(* IEC 61131-3 sources: sphere-usecases/sector-energy/olmsted-hydro/implementations/openplc/st/legacy, 2 files *)

(* ---- ps_hydro_controller.st ---- *)
(*
 * SPHERE Power Systems - Generic Hydro Station Controller
 * IEC 61131-3 Structured Text for OpenPLC
 *
 * Control state machine for hydro power generation:
 *   IDLE -> STARTUP -> RUNNING -> SHUTDOWN -> IDLE
 *                  \-> TRIPPED (on any trip) -> IDLE (after reset)
 *
 * This program runs on the CONTROLLER PLC and implements:
 *   - State machine for unit operation
 *   - Permissive checks for startup
 *   - Power tracking via gate modulation (P-control)
 *   - Trip detection and response
 *   - Mismatch alarm generation
 *
 * Inputs (from HMI):
 *   - Start, Stop, Reset commands (%IX0.0-0.2)
 *   - Mode Auto, Run Enable (%IX0.3-0.4)
 *
 * Inputs (from Simulator via bridge):
 *   - Gate position, sensors (%IW70-77)
 *   - Breaker/Spill status (%IX2.0-2.1)
 *
 * Outputs (to Simulator via bridge):
 *   - Gate command (%QW100)
 *   - Breaker/Spill commands (%QX5.0-5.1)
 *
 * Outputs (to HMI):
 *   - State indicators (%QX7.0-7.5)
 *   - Trip indicators (%QX8.0-8.3)
 *   - Alarm indicators (%QX9.0-9.2)
 *)

(* ═══════════════════════════════════════════════════════════════════════════
   GLOBAL VARIABLES - I/O MAPPING
   ═══════════════════════════════════════════════════════════════════════════ *)
VAR_GLOBAL
    (* HMI Inputs *)
    in_Start_Cmd AT %IX0.0 : BOOL;      (* Start pushbutton *)
    in_Stop_Cmd AT %IX0.1 : BOOL;       (* Stop pushbutton *)
    in_Reset_Cmd AT %IX0.2 : BOOL;      (* Trip reset pushbutton *)
    in_Mode_Auto AT %IX0.3 : BOOL;      (* Auto mode enable *)
    in_Run_Enable AT %IX0.4 : BOOL;     (* Run permissive *)

    (* Power setpoint - could come from HMI or external *)
    in_Power_Setpoint AT %IW60 : INT;   (* 0-1000 = 0-100 MW *)

    (* Process Inputs from Simulator (via bridge) *)
    in_Gate_Pos AT %IW70 : INT;         (* Gate position 0-1000 = 0-100% *)
    in_Res_Level AT %IW71 : INT;        (* Reservoir level 0-3000 = 0-30.00 m *)
    in_Head AT %IW72 : INT;             (* Head 0-1500 = 0-150.0 m *)
    in_Flow AT %IW73 : INT;             (* Flow 0-1500 = 0-150.0 m3/s *)
    in_Pressure AT %IW74 : INT;         (* Pressure kPa *)
    in_Speed_Pct AT %IW75 : INT;        (* Speed 0-1500 = 0-150.0% *)
    in_Freq_Hz AT %IW76 : INT;          (* Frequency 5500-6500 = 55-65 Hz *)
    in_Power_MW AT %IW77 : INT;         (* Power 0-1000 = 0-100 MW *)

    in_Breaker_Sts AT %IX2.0 : BOOL;    (* Breaker closed status *)
    in_Spill_Sts AT %IX2.1 : BOOL;      (* Spillway open status *)

    (* Actuator Outputs to Simulator (via bridge) *)
    out_Gate_Cmd AT %QW100 : INT;       (* Gate command 0-1000 = 0-100% *)
    out_Power_Setpoint AT %QW101 : INT; (* Power setpoint passthrough *)
    out_Breaker_Cmd AT %QX5.0 : BOOL;   (* Breaker close command *)
    out_Spill_Cmd AT %QX5.1 : BOOL;     (* Spillway open command *)

    (* State Outputs to HMI *)
    out_State_Idle AT %QX7.0 : BOOL;
    out_State_Startup AT %QX7.1 : BOOL;
    out_State_Running AT %QX7.2 : BOOL;
    out_State_Shutdown AT %QX7.3 : BOOL;
    out_State_Tripped AT %QX7.4 : BOOL;
    out_Permissives_Ready AT %QX7.5 : BOOL;

    (* Trip Outputs *)
    out_Trip_Overspeed AT %QX8.0 : BOOL;
    out_Trip_Overpressure AT %QX8.1 : BOOL;
    out_Trip_LowHead AT %QX8.2 : BOOL;
    out_Trip_Manual AT %QX8.3 : BOOL;

    (* Alarm Outputs *)
    out_Alarm_GateMismatch AT %QX9.0 : BOOL;
    out_Alarm_BreakerMismatch AT %QX9.1 : BOOL;
    out_Alarm_LowLevel AT %QX9.2 : BOOL;
END_VAR

(* ═══════════════════════════════════════════════════════════════════════════
   MAIN PROGRAM
   ═══════════════════════════════════════════════════════════════════════════ *)
PROGRAM HydroController
VAR
    (* ─── State Machine ──────────────────────────────────────────────────── *)
    State : INT := 0;                   (* 0=IDLE, 1=STARTUP, 2=RUNNING, 3=SHUTDOWN, 4=TRIPPED *)
    STATE_IDLE : INT := 0;
    STATE_STARTUP : INT := 1;
    STATE_RUNNING : INT := 2;
    STATE_SHUTDOWN : INT := 3;
    STATE_TRIPPED : INT := 4;

    (* ─── Permissives ────────────────────────────────────────────────────── *)
    Perm_Level_OK : BOOL := FALSE;      (* Reservoir level adequate *)
    Perm_Head_OK : BOOL := FALSE;       (* Head above minimum *)
    Perm_No_Trips : BOOL := FALSE;      (* No active trips *)
    Perm_Run_Enable : BOOL := FALSE;    (* Operator run enable *)
    All_Permissives : BOOL := FALSE;    (* Combined permissive *)

    (* ─── Trip Latches ───────────────────────────────────────────────────── *)
    Trip_Overspeed_Latch : BOOL := FALSE;
    Trip_Overpressure_Latch : BOOL := FALSE;
    Trip_LowHead_Latch : BOOL := FALSE;
    Trip_Manual_Latch : BOOL := FALSE;
    Any_Trip : BOOL := FALSE;

    (* ─── Control Parameters ─────────────────────────────────────────────── *)
    No_Load_Gate_Pct : REAL := 5.0;     (* Gate position for no-load sync *)
    Sync_Speed_Low : REAL := 99.0;      (* Min speed for sync % *)
    Sync_Speed_High : REAL := 101.0;    (* Max speed for sync % *)
    Min_Power_MW : REAL := 1.0;         (* Min power before breaker open *)
    Kp_Gate : REAL := 2.0;              (* Power control gain *)
    Gate_Shutdown_Rate : REAL := 5.0;   (* %/sample during shutdown *)
    Gate_Emerg_Rate : REAL := 20.0;     (* %/sample during trip *)

    (* ─── Trip Thresholds ────────────────────────────────────────────────── *)
    Overspeed_Trip_Pct : REAL := 110.0;
    Overpressure_Trip_kPa : REAL := 1500.0;
    Min_Head_m : REAL := 10.0;
    Low_Level_m : REAL := 8.0;          (* Alarm threshold *)

    (* ─── Mismatch Alarm Parameters ──────────────────────────────────────── *)
    Gate_Mismatch_Pct : REAL := 5.0;    (* Alarm if error > 5% *)
    Gate_Mismatch_Delay : INT := 50;    (* 5 sec at 100ms cycle *)
    Breaker_Mismatch_Delay : INT := 5;  (* 0.5 sec *)
    Gate_Mismatch_Timer : INT := 0;
    Breaker_Mismatch_Timer : INT := 0;

    (* ─── Process Values (scaled) ────────────────────────────────────────── *)
    Gate_Pos_Pct : REAL;
    Gate_Cmd_Pct : REAL := 0.0;
    Res_Level_m : REAL;
    Head_m : REAL;
    Flow_m3s : REAL;
    Pressure_kPa : REAL;
    Speed_Pct : REAL;
    Freq_Hz : REAL;
    Power_MW : REAL;
    Power_Setpoint_MW : REAL;

    (* ─── Control Calculations ───────────────────────────────────────────── *)
    Power_Error : REAL;
    Gate_Adjustment : REAL;

    (* ─── Edge Detection ─────────────────────────────────────────────────── *)
    Start_Cmd_Prev : BOOL := FALSE;
    Stop_Cmd_Prev : BOOL := FALSE;
    Reset_Cmd_Prev : BOOL := FALSE;
    Start_Rising : BOOL := FALSE;
    Stop_Rising : BOOL := FALSE;
    Reset_Rising : BOOL := FALSE;
END_VAR

(* ═══════════════════════════════════════════════════════════════════════════
   CONTROL LOGIC
   ═══════════════════════════════════════════════════════════════════════════ *)

(* ─── 1. SCALE INPUTS ─────────────────────────────────────────────────────── *)
Gate_Pos_Pct := INT_TO_REAL(in_Gate_Pos) / 10.0;
Res_Level_m := INT_TO_REAL(in_Res_Level) / 100.0;
Head_m := INT_TO_REAL(in_Head) / 10.0;
Flow_m3s := INT_TO_REAL(in_Flow) / 10.0;
Pressure_kPa := INT_TO_REAL(in_Pressure);
Speed_Pct := INT_TO_REAL(in_Speed_Pct) / 10.0;
Freq_Hz := INT_TO_REAL(in_Freq_Hz) / 100.0;
Power_MW := INT_TO_REAL(in_Power_MW) / 10.0;
Power_Setpoint_MW := INT_TO_REAL(in_Power_Setpoint) / 10.0;

(* ─── 2. EDGE DETECTION FOR COMMANDS ──────────────────────────────────────── *)
Start_Rising := in_Start_Cmd AND NOT Start_Cmd_Prev;
Stop_Rising := in_Stop_Cmd AND NOT Stop_Cmd_Prev;
Reset_Rising := in_Reset_Cmd AND NOT Reset_Cmd_Prev;
Start_Cmd_Prev := in_Start_Cmd;
Stop_Cmd_Prev := in_Stop_Cmd;
Reset_Cmd_Prev := in_Reset_Cmd;

(* ─── 3. TRIP DETECTION ───────────────────────────────────────────────────── *)
(* Check trip conditions and latch *)
IF Speed_Pct > Overspeed_Trip_Pct THEN
    Trip_Overspeed_Latch := TRUE;
END_IF;

IF Pressure_kPa > Overpressure_Trip_kPa THEN
    Trip_Overpressure_Latch := TRUE;
END_IF;

IF Head_m < Min_Head_m AND State = STATE_RUNNING THEN
    Trip_LowHead_Latch := TRUE;
END_IF;

(* Manual trip via Stop during running with specific pattern *)
(* For now, no separate manual trip - Stop just initiates shutdown *)

(* Combined trip check *)
Any_Trip := Trip_Overspeed_Latch OR Trip_Overpressure_Latch OR
            Trip_LowHead_Latch OR Trip_Manual_Latch;

(* ─── 4. PERMISSIVE CHECKS ────────────────────────────────────────────────── *)
Perm_Level_OK := Res_Level_m > Low_Level_m;
Perm_Head_OK := Head_m >= Min_Head_m;
Perm_No_Trips := NOT Any_Trip;
Perm_Run_Enable := in_Run_Enable;

All_Permissives := Perm_Level_OK AND Perm_Head_OK AND
                   Perm_No_Trips AND Perm_Run_Enable;

(* ─── 5. STATE MACHINE ────────────────────────────────────────────────────── *)
CASE State OF
    (* ═══ IDLE STATE ═══ *)
    0: (* STATE_IDLE *)
        (* Outputs: gate closed, breaker open *)
        Gate_Cmd_Pct := 0.0;
        out_Breaker_Cmd := FALSE;
        out_Spill_Cmd := FALSE;

        (* Transitions *)
        IF Start_Rising AND All_Permissives THEN
            State := STATE_STARTUP;
        END_IF;

    (* ═══ STARTUP STATE ═══ *)
    1: (* STATE_STARTUP *)
        (* Ramp gate to no-load position *)
        IF Gate_Cmd_Pct < No_Load_Gate_Pct THEN
            Gate_Cmd_Pct := Gate_Cmd_Pct + 1.0;  (* Ramp up 1%/cycle *)
        ELSE
            Gate_Cmd_Pct := No_Load_Gate_Pct;
        END_IF;

        (* Check for sync conditions *)
        IF Speed_Pct >= Sync_Speed_Low AND Speed_Pct <= Sync_Speed_High THEN
            (* Close breaker when speed is in sync range *)
            out_Breaker_Cmd := TRUE;

            (* Transition to running when breaker closes *)
            IF in_Breaker_Sts THEN
                State := STATE_RUNNING;
            END_IF;
        END_IF;

        (* Trip handling *)
        IF Any_Trip THEN
            State := STATE_TRIPPED;
        END_IF;

        (* Stop command *)
        IF Stop_Rising THEN
            State := STATE_SHUTDOWN;
        END_IF;

    (* ═══ RUNNING STATE ═══ *)
    2: (* STATE_RUNNING *)
        (* Power tracking via P-control *)
        Power_Error := Power_Setpoint_MW - Power_MW;
        Gate_Adjustment := Kp_Gate * Power_Error;

        (* Apply adjustment with limits *)
        Gate_Cmd_Pct := Gate_Cmd_Pct + Gate_Adjustment;

        (* Clamp gate command *)
        IF Gate_Cmd_Pct < 0.0 THEN Gate_Cmd_Pct := 0.0; END_IF;
        IF Gate_Cmd_Pct > 100.0 THEN Gate_Cmd_Pct := 100.0; END_IF;

        (* Breaker stays closed *)
        out_Breaker_Cmd := TRUE;

        (* Trip handling - immediate transition *)
        IF Any_Trip THEN
            State := STATE_TRIPPED;
        END_IF;

        (* Stop command - normal shutdown *)
        IF Stop_Rising THEN
            State := STATE_SHUTDOWN;
        END_IF;

    (* ═══ SHUTDOWN STATE ═══ *)
    3: (* STATE_SHUTDOWN *)
        (* Ramp gate down *)
        Gate_Cmd_Pct := Gate_Cmd_Pct - Gate_Shutdown_Rate;
        IF Gate_Cmd_Pct < 0.0 THEN
            Gate_Cmd_Pct := 0.0;
        END_IF;

        (* Open breaker when power is low enough *)
        IF Power_MW < Min_Power_MW THEN
            out_Breaker_Cmd := FALSE;
        END_IF;

        (* Transition to idle when gate closed and breaker open *)
        IF Gate_Cmd_Pct <= 0.0 AND NOT in_Breaker_Sts THEN
            State := STATE_IDLE;
        END_IF;

        (* Trip can still occur during shutdown *)
        IF Any_Trip THEN
            State := STATE_TRIPPED;
        END_IF;

    (* ═══ TRIPPED STATE ═══ *)
    4: (* STATE_TRIPPED *)
        (* Emergency actions *)
        out_Breaker_Cmd := FALSE;           (* Open breaker immediately *)

        (* Fast gate close *)
        Gate_Cmd_Pct := Gate_Cmd_Pct - Gate_Emerg_Rate;
        IF Gate_Cmd_Pct < 0.0 THEN
            Gate_Cmd_Pct := 0.0;
        END_IF;

        (* Open spillway on overspeed to dump water *)
        IF Trip_Overspeed_Latch THEN
            out_Spill_Cmd := TRUE;
        END_IF;

        (* Reset handling - only when gate closed and breaker open *)
        IF Reset_Rising AND Gate_Cmd_Pct <= 0.0 AND NOT in_Breaker_Sts THEN
            (* Clear all trip latches *)
            Trip_Overspeed_Latch := FALSE;
            Trip_Overpressure_Latch := FALSE;
            Trip_LowHead_Latch := FALSE;
            Trip_Manual_Latch := FALSE;

            (* Close spillway *)
            out_Spill_Cmd := FALSE;

            (* Return to idle *)
            State := STATE_IDLE;
        END_IF;

END_CASE;

(* ─── 6. MISMATCH ALARM LOGIC ─────────────────────────────────────────────── *)
(* Gate mismatch alarm *)
IF ABS(Gate_Cmd_Pct - Gate_Pos_Pct) > Gate_Mismatch_Pct THEN
    Gate_Mismatch_Timer := Gate_Mismatch_Timer + 1;
    IF Gate_Mismatch_Timer >= Gate_Mismatch_Delay THEN
        out_Alarm_GateMismatch := TRUE;
    END_IF;
ELSE
    Gate_Mismatch_Timer := 0;
    out_Alarm_GateMismatch := FALSE;
END_IF;

(* Breaker mismatch alarm *)
IF out_Breaker_Cmd <> in_Breaker_Sts THEN
    Breaker_Mismatch_Timer := Breaker_Mismatch_Timer + 1;
    IF Breaker_Mismatch_Timer >= Breaker_Mismatch_Delay THEN
        out_Alarm_BreakerMismatch := TRUE;
    END_IF;
ELSE
    Breaker_Mismatch_Timer := 0;
    out_Alarm_BreakerMismatch := FALSE;
END_IF;

(* Low level alarm *)
out_Alarm_LowLevel := Res_Level_m < Low_Level_m;

(* ─── 7. WRITE OUTPUTS ────────────────────────────────────────────────────── *)
(* Scale and write gate command *)
out_Gate_Cmd := REAL_TO_INT(Gate_Cmd_Pct * 10.0);

(* Pass through power setpoint *)
out_Power_Setpoint := in_Power_Setpoint;

(* State indicators *)
out_State_Idle := (State = STATE_IDLE);
out_State_Startup := (State = STATE_STARTUP);
out_State_Running := (State = STATE_RUNNING);
out_State_Shutdown := (State = STATE_SHUTDOWN);
out_State_Tripped := (State = STATE_TRIPPED);
out_Permissives_Ready := All_Permissives;

(* Trip indicators *)
out_Trip_Overspeed := Trip_Overspeed_Latch;
out_Trip_Overpressure := Trip_Overpressure_Latch;
out_Trip_LowHead := Trip_LowHead_Latch;
out_Trip_Manual := Trip_Manual_Latch;

END_PROGRAM

(* ---- ps_hydro_simulator.st ---- *)
(*
 * SPHERE Power Systems - Generic Hydro Station Simulator
 * IEC 61131-3 Structured Text for OpenPLC
 *
 * Physics model for hydro power generation:
 *   Reservoir -> Penstock -> Wicket Gate -> Turbine -> Generator -> Breaker -> Grid
 *
 * This program runs on the SIMULATOR PLC and models:
 *   - Reservoir mass balance with head calculation
 *   - Penstock flow dynamics (1st-order lag)
 *   - Wicket gate actuator with slew limits
 *   - Turbine/generator power conversion
 *   - Breaker dynamics
 *   - Trip condition detection
 *
 * Inputs (from Controller via bridge):
 *   - Gate command (%IW200)
 *   - Breaker command (%IX3.0)
 *   - Spill command (%IX3.1)
 *
 * Outputs (to Controller via bridge):
 *   - Gate position (%QW300)
 *   - Reservoir level, head, flow, pressure, speed, freq, power (%QW301-307)
 *   - Breaker status, spill status (%QX40.0-40.1)
 *)

(* ═══════════════════════════════════════════════════════════════════════════
   GLOBAL VARIABLES - I/O MAPPING
   ═══════════════════════════════════════════════════════════════════════════ *)
VAR_GLOBAL
    (* Inputs from Controller (via bridge) *)
    in_Gate_Cmd AT %IW200 : INT;        (* Gate command 0-1000 = 0-100% *)
    in_Breaker_Cmd AT %IX3.0 : BOOL;    (* Breaker close command *)
    in_Spill_Cmd AT %IX3.1 : BOOL;      (* Spillway open command *)

    (* Outputs to Controller (via bridge) *)
    out_Gate_Pos AT %QW300 : INT;       (* Gate position 0-1000 = 0-100% *)
    out_Res_Level AT %QW301 : INT;      (* Reservoir level 0-3000 = 0-30.00 m *)
    out_Head AT %QW302 : INT;           (* Head 0-1500 = 0-150.0 m *)
    out_Flow AT %QW303 : INT;           (* Flow 0-1500 = 0-150.0 m3/s *)
    out_Pressure AT %QW304 : INT;       (* Pressure 0-2000 kPa *)
    out_Speed_Pct AT %QW305 : INT;      (* Speed 0-1500 = 0-150.0% *)
    out_Freq_Hz AT %QW306 : INT;        (* Frequency 5500-6500 = 55.00-65.00 Hz *)
    out_Power_MW AT %QW307 : INT;       (* Power 0-1000 = 0-100.0 MW *)

    out_Breaker_Sts AT %QX40.0 : BOOL;  (* Breaker closed status *)
    out_Spill_Sts AT %QX40.1 : BOOL;    (* Spillway open status *)
END_VAR

(* ═══════════════════════════════════════════════════════════════════════════
   MAIN PROGRAM
   ═══════════════════════════════════════════════════════════════════════════ *)
PROGRAM HydroSimulator
VAR
    (* ─── Physical Parameters (from profile) ─────────────────────────────── *)
    (* Reservoir *)
    Res_Area_m2 : REAL := 10000.0;      (* Reservoir surface area *)
    Res_Level_m : REAL := 20.0;         (* Current reservoir level *)
    Res_Inflow_m3s : REAL := 50.0;      (* Natural inflow *)
    Res_Min_m : REAL := 5.0;            (* Minimum operating level *)
    Res_Max_m : REAL := 25.0;           (* Maximum level *)
    Tailwater_m : REAL := 0.0;          (* Tailwater elevation *)

    (* Penstock *)
    Penstock_Tau_sec : REAL := 5.0;     (* Flow inertia time constant *)
    Static_Head_m : REAL := 100.0;      (* Reference static head *)

    (* Turbine *)
    Q_Max_m3s : REAL := 100.0;          (* Maximum flow capacity *)
    Eta_Turbine : REAL := 0.90;         (* Turbine efficiency *)
    K_Q : REAL := 10.0;                 (* Flow coefficient *)

    (* Generator *)
    Eta_Gen : REAL := 0.97;             (* Generator efficiency *)
    P_Rated_MW : REAL := 80.0;          (* Rated power *)
    Inertia_H : REAL := 4.0;            (* Inertia constant (seconds) *)
    Sync_Speed_Pct : REAL := 100.0;     (* Synchronous speed reference *)

    (* Gate actuator *)
    Gate_Travel_sec : REAL := 10.0;     (* Full stroke time *)
    Gate_Slew_Max : REAL := 10.0;       (* Max slew rate %/s *)
    Gate_Tau_sec : REAL := 1.0;         (* Servo time constant *)
    Gate_Emerg_sec : REAL := 3.0;       (* Emergency close time *)

    (* Breaker *)
    Breaker_Open_sec : REAL := 0.06;    (* Open time *)
    Breaker_Close_sec : REAL := 0.05;   (* Close time *)

    (* Spillway *)
    Spill_Open_sec : REAL := 5.0;       (* Spillway open time *)

    (* Physical constants *)
    RHO : REAL := 1000.0;               (* Water density kg/m3 *)
    G : REAL := 9.81;                   (* Gravity m/s2 *)

    (* ─── State Variables ────────────────────────────────────────────────── *)
    Gate_Pos_Pct : REAL := 0.0;         (* Actual gate position % *)
    Gate_Vel : REAL := 0.0;             (* Gate velocity %/s *)
    Flow_m3s : REAL := 0.0;             (* Actual flow rate *)
    Flow_Target_m3s : REAL := 0.0;      (* Target flow (gate opening) *)
    Head_m : REAL := 100.0;             (* Net hydraulic head *)
    Pressure_kPa : REAL := 981.0;       (* Penstock pressure *)
    Speed_Pct : REAL := 0.0;            (* Turbine speed % of sync *)
    Freq_Hz : REAL := 0.0;              (* Electrical frequency *)
    P_Mech_MW : REAL := 0.0;            (* Mechanical power *)
    P_Elec_MW : REAL := 0.0;            (* Electrical power *)

    Breaker_Closed : BOOL := FALSE;     (* Breaker state *)
    Breaker_Timer : REAL := 0.0;        (* Breaker transition timer *)
    Spill_Open : BOOL := FALSE;         (* Spillway state *)
    Spill_Timer : REAL := 0.0;          (* Spillway transition timer *)

    (* ─── Intermediate Calculations ──────────────────────────────────────── *)
    Gate_Cmd_Pct : REAL;                (* Commanded gate position % *)
    Gate_Error : REAL;                  (* Gate position error *)
    dQ_dt : REAL;                       (* Flow rate of change *)
    dLevel_dt : REAL;                   (* Level rate of change *)
    dSpeed_dt : REAL;                   (* Speed rate of change *)
    P_Load_MW : REAL;                   (* Grid load (when connected) *)
    Spill_Flow_m3s : REAL;              (* Spillway discharge *)

    (* ─── Timing ─────────────────────────────────────────────────────────── *)
    DT : REAL := 0.1;                   (* Simulation timestep (100ms) *)

    (* ─── Trip Detection ─────────────────────────────────────────────────── *)
    Overspeed : BOOL := FALSE;
    Overpressure : BOOL := FALSE;
    LowHead : BOOL := FALSE;
END_VAR

(* ═══════════════════════════════════════════════════════════════════════════
   SIMULATION LOGIC
   ═══════════════════════════════════════════════════════════════════════════ *)

(* ─── 1. PROCESS INPUTS ───────────────────────────────────────────────────── *)
(* Convert scaled integer inputs to engineering units *)
Gate_Cmd_Pct := INT_TO_REAL(in_Gate_Cmd) / 10.0;  (* 0-1000 -> 0-100% *)

(* Clamp command to valid range *)
IF Gate_Cmd_Pct < 0.0 THEN Gate_Cmd_Pct := 0.0; END_IF;
IF Gate_Cmd_Pct > 100.0 THEN Gate_Cmd_Pct := 100.0; END_IF;

(* ─── 2. GATE ACTUATOR DYNAMICS ───────────────────────────────────────────── *)
(* First-order servo response with slew limiting *)
Gate_Error := Gate_Cmd_Pct - Gate_Pos_Pct;
Gate_Vel := Gate_Error / Gate_Tau_sec;

(* Apply slew rate limits *)
IF Gate_Vel > Gate_Slew_Max THEN
    Gate_Vel := Gate_Slew_Max;
ELSIF Gate_Vel < -Gate_Slew_Max THEN
    Gate_Vel := -Gate_Slew_Max;
END_IF;

(* Integrate gate position *)
Gate_Pos_Pct := Gate_Pos_Pct + Gate_Vel * DT;

(* Clamp to physical limits *)
IF Gate_Pos_Pct < 0.0 THEN Gate_Pos_Pct := 0.0; END_IF;
IF Gate_Pos_Pct > 100.0 THEN Gate_Pos_Pct := 100.0; END_IF;

(* ─── 3. RESERVOIR MASS BALANCE ───────────────────────────────────────────── *)
(* Calculate spillway flow if open *)
IF Spill_Open THEN
    (* Simple spillway model: proportional to level above threshold *)
    IF Res_Level_m > 22.0 THEN
        Spill_Flow_m3s := 20.0 * (Res_Level_m - 22.0);
    ELSE
        Spill_Flow_m3s := 0.0;
    END_IF;
ELSE
    Spill_Flow_m3s := 0.0;
END_IF;

(* Mass balance: dV/dt = Q_in - Q_turbine - Q_spill *)
dLevel_dt := (Res_Inflow_m3s - Flow_m3s - Spill_Flow_m3s) / Res_Area_m2;
Res_Level_m := Res_Level_m + dLevel_dt * DT;

(* Clamp reservoir level *)
IF Res_Level_m < 0.0 THEN Res_Level_m := 0.0; END_IF;
IF Res_Level_m > Res_Max_m THEN Res_Level_m := Res_Max_m; END_IF;

(* Calculate net head: H = reservoir_level - tailwater *)
Head_m := Res_Level_m + Static_Head_m - Tailwater_m;
IF Head_m < 0.0 THEN Head_m := 0.0; END_IF;

(* ─── 4. PENSTOCK FLOW DYNAMICS ───────────────────────────────────────────── *)
(* Target flow based on gate opening and head *)
(* Q = k_q * (gate_pos/100) * sqrt(H) *)
IF Head_m > 0.0 THEN
    Flow_Target_m3s := K_Q * (Gate_Pos_Pct / 100.0) * SQRT(Head_m);
ELSE
    Flow_Target_m3s := 0.0;
END_IF;

(* Limit to maximum flow *)
IF Flow_Target_m3s > Q_Max_m3s THEN
    Flow_Target_m3s := Q_Max_m3s;
END_IF;

(* First-order lag for flow inertia: dQ/dt = (Q_target - Q) / tau *)
dQ_dt := (Flow_Target_m3s - Flow_m3s) / Penstock_Tau_sec;
Flow_m3s := Flow_m3s + dQ_dt * DT;

(* Clamp flow *)
IF Flow_m3s < 0.0 THEN Flow_m3s := 0.0; END_IF;

(* Calculate penstock pressure: P = rho * g * H *)
Pressure_kPa := RHO * G * Head_m / 1000.0;

(* Check for water hammer (rapid flow change) *)
IF ABS(dQ_dt) > 20.0 THEN
    (* Approximate pressure surge *)
    Pressure_kPa := Pressure_kPa * 1.5;
END_IF;

(* ─── 5. TURBINE/GENERATOR DYNAMICS ───────────────────────────────────────── *)
(* Mechanical power: P_mech = rho * g * Q * H * eta_t *)
P_Mech_MW := RHO * G * Flow_m3s * Head_m * Eta_Turbine / 1000000.0;

(* Speed dynamics depend on breaker state *)
IF Breaker_Closed THEN
    (* Connected to grid - speed locked to sync *)
    Speed_Pct := 100.0;
    Freq_Hz := 60.0;

    (* Electrical power = min(mechanical power * eta_g, rated) *)
    P_Elec_MW := P_Mech_MW * Eta_Gen;
    IF P_Elec_MW > P_Rated_MW THEN
        P_Elec_MW := P_Rated_MW;
    END_IF;
ELSE
    (* Offline - speed determined by turbine power vs losses *)
    (* Simplified: speed rises with flow, falls with friction *)
    IF Flow_m3s > 0.1 THEN
        (* Accelerating: dSpeed/dt proportional to (torque - friction) *)
        dSpeed_dt := (P_Mech_MW / (P_Rated_MW * 0.1) - Speed_Pct / 50.0) / Inertia_H;
        Speed_Pct := Speed_Pct + dSpeed_dt * DT;
    ELSE
        (* Decelerating: coast down *)
        dSpeed_dt := -Speed_Pct / (Inertia_H * 10.0);
        Speed_Pct := Speed_Pct + dSpeed_dt * DT;
    END_IF;

    (* Clamp speed *)
    IF Speed_Pct < 0.0 THEN Speed_Pct := 0.0; END_IF;
    IF Speed_Pct > 150.0 THEN Speed_Pct := 150.0; END_IF;

    (* Frequency proportional to speed *)
    Freq_Hz := 60.0 * Speed_Pct / 100.0;

    (* No electrical power when offline *)
    P_Elec_MW := 0.0;
END_IF;

(* ─── 6. BREAKER DYNAMICS ─────────────────────────────────────────────────── *)
IF in_Breaker_Cmd AND NOT Breaker_Closed THEN
    (* Close command received - start closing *)
    Breaker_Timer := Breaker_Timer + DT;
    IF Breaker_Timer >= Breaker_Close_sec THEN
        (* Check sync conditions before closing *)
        IF Speed_Pct >= 99.0 AND Speed_Pct <= 101.0 THEN
            Breaker_Closed := TRUE;
        END_IF;
        Breaker_Timer := 0.0;
    END_IF;
ELSIF NOT in_Breaker_Cmd AND Breaker_Closed THEN
    (* Open command received - start opening *)
    Breaker_Timer := Breaker_Timer + DT;
    IF Breaker_Timer >= Breaker_Open_sec THEN
        Breaker_Closed := FALSE;
        Breaker_Timer := 0.0;
    END_IF;
ELSE
    Breaker_Timer := 0.0;
END_IF;

(* ─── 7. SPILLWAY DYNAMICS ────────────────────────────────────────────────── *)
IF in_Spill_Cmd AND NOT Spill_Open THEN
    Spill_Timer := Spill_Timer + DT;
    IF Spill_Timer >= Spill_Open_sec THEN
        Spill_Open := TRUE;
        Spill_Timer := 0.0;
    END_IF;
ELSIF NOT in_Spill_Cmd AND Spill_Open THEN
    Spill_Timer := Spill_Timer + DT;
    IF Spill_Timer >= Spill_Open_sec THEN
        Spill_Open := FALSE;
        Spill_Timer := 0.0;
    END_IF;
ELSE
    Spill_Timer := 0.0;
END_IF;

(* ─── 8. TRIP CONDITION DETECTION ─────────────────────────────────────────── *)
(* These are informational - actual trip logic is in controller *)
Overspeed := Speed_Pct > 110.0;
Overpressure := Pressure_kPa > (RHO * G * Static_Head_m / 1000.0) * 1.5;
LowHead := Head_m < 10.0;

(* ─── 9. WRITE OUTPUTS ────────────────────────────────────────────────────── *)
(* Convert engineering units to scaled integers for Modbus *)
out_Gate_Pos := REAL_TO_INT(Gate_Pos_Pct * 10.0);           (* 0-100% -> 0-1000 *)
out_Res_Level := REAL_TO_INT(Res_Level_m * 100.0);          (* 0-30m -> 0-3000 *)
out_Head := REAL_TO_INT(Head_m * 10.0);                     (* 0-150m -> 0-1500 *)
out_Flow := REAL_TO_INT(Flow_m3s * 10.0);                   (* 0-150m3/s -> 0-1500 *)
out_Pressure := REAL_TO_INT(Pressure_kPa);                  (* kPa direct *)
out_Speed_Pct := REAL_TO_INT(Speed_Pct * 10.0);             (* 0-150% -> 0-1500 *)
out_Freq_Hz := REAL_TO_INT(Freq_Hz * 100.0);                (* 55-65Hz -> 5500-6500 *)
out_Power_MW := REAL_TO_INT(P_Elec_MW * 10.0);              (* 0-100MW -> 0-1000 *)

out_Breaker_Sts := Breaker_Closed;
out_Spill_Sts := Spill_Open;

END_PROGRAM
